// ==============================================================================
// FC_RouteFSM - Керування маршрутом (Mailbox Pattern v3.9)
// ==============================================================================
// Версія: 3.9.2
// Дата: 2026-02-27
// ==============================================================================
// ГАРАНТІЇ ЗУПИНКИ:
//   Нормальний STOP_OP:
//     STOPPING: CMD_STOP кожен цикл → STS_STOPPING→STS_IDLE →
//     allStopped → CMD_RELEASE_OWNER (ARB_OK) → ABORTED ✓
//
//   Аварія під час зупинки (STOPPING):
//     STS_FAULT → allStopped (FAULT рахується) →
//     CMD_RELEASE_OWNER (ARB_OK, FAULT дозволено) → ABORTED ✓
//
//   Enable_OK знімається під час зупинки (STOPPING):
//     STS_DISABLED + OwnerCur=NONE (механізм сам скинув) → allStopped →
//     CMD_RELEASE_OWNER → ARB_OWNER_BUSY (dummyOk) → ABORTED ✓
//
//   GlobalSafetyStop (механізм у STS_RUNNING):
//     CMD_STOP → Mechs[slot].Cmd=CMD_STOP → механізм → STS_STOPPING
//     CMD_RELEASE_OWNER → ARB_WRONG_STATUS (ще не IDLE) → ABORTED
//     Retry у ABORTED: STS_STOPPING→STS_IDLE → ARB_OK → OwnerCur=NONE ✓
//     (якщо апаратна безпека вбила живлення → STS_FAULT → ARB_OK ✓)
//
// АРХІТЕКТУРА:
//   FC_RouteFSM    — логіка переходів, послідовність кроків
//   FC_ArbiterMech — захоплення ownership, запис команди
//   FC_Noria/...   — виконання команди, зміна Status, аварії
//   FC_Route_Supervisor — Mailbox→RouteExecutor, виклик FSM, cleanup
// ==============================================================================

FUNCTION "FC_RouteFSM" : Void
{ S7_Optimized_Access := 'TRUE' }
VERSION : 3.7

VAR_INPUT
    RouteIdx          : USINT;            // ID маршруту (1..12)
    Cmd               : "UDT_RouteCmd";   // Команда та кроки маршруту
END_VAR

VAR_IN_OUT
    Mechs : ARRAY[0.."MECHS_COUNT"] OF "UDT_BaseMechanism";
    Fsm   : "UDT_RouteFsm";
END_VAR

VAR_OUTPUT
    Sts : "UDT_RouteStatus";
END_VAR

VAR_TEMP
    timeElapsed : BOOL;   // проміжний результат FC_TimeElapsedMs
    elapsedMs   : DINT;   // допоміжний вихід FC_TimeElapsedMs (ігнорується)
    nowTck      : DINT;   // допоміжний вихід FC_TimeElapsedMs (ігнорується)
    doAdvance   : BOOL;   // TRUE = виконати advance у STOPPING (після Phase A або Phase B)
END_VAR

BEGIN

    // =========================================================
    // Edge detection команд маршруту
    // =========================================================
    Fsm.startEdge  := (Cmd.RC_Cmd = "RT_CMD_START")   AND (Fsm.lastCmd <> "RT_CMD_START");
    Fsm.stopOpEdge := (Cmd.RC_Cmd = "RT_CMD_STOP_OP") AND (Fsm.lastCmd <> "RT_CMD_STOP_OP");
    Fsm.lastCmd    := Cmd.RC_Cmd;

    // =========================================================
    // Кількість кроків (з обмеженням)
    // =========================================================
    Fsm.stepCnt := USINT_TO_INT(Cmd.RC_StepCount);
    IF Fsm.stepCnt < 1  THEN Fsm.stepCnt := 1;  END_IF;
    IF Fsm.stepCnt > "ROUTE_MAX_STEPS" THEN Fsm.stepCnt := "ROUTE_MAX_STEPS"; END_IF;

    // Захист від неініціалізованого стану
    IF Fsm.RF_State = 0 THEN
        Fsm.RF_State := "ROUTE_STS_IDLE";
    END_IF;

    // =========================================================
    // Сканування механізмів: аварії та LocalManual
    // =========================================================
    Fsm.anyFault  := FALSE;
    Fsm.anyLocal  := FALSE;
    Fsm.safetyHit := FALSE;

    IF Fsm.stepCnt > 0 THEN
        FOR Fsm.i := 1 TO Fsm.stepCnt DO
            Fsm.slot := Cmd.RC_Steps[Fsm.i].RS_Slot;
            IF Fsm.slot > "MECHS_COUNT" THEN CONTINUE; END_IF;

            IF Mechs[Fsm.slot].FLTCode <> 0 THEN
                Fsm.anyFault := TRUE;
            END_IF;

            IF GlobalLocalManual OR Mechs[Fsm.slot].LocalManual THEN
                Fsm.anyLocal := TRUE;
            END_IF;

            IF Fsm.anyFault AND Fsm.anyLocal THEN EXIT; END_IF;
        END_FOR;
    END_IF;

    // =========================================================
    // АВАРІЙНА ЗУПИНКА (GlobalSafetyStop) — найвищий пріоритет
    // =========================================================
    // Послідовність для кожного механізму:
    //   1. CMD_STOP       — наказ зупинитись негайно (незалежно від послідовності)
    //                       ARB_OK → Mechs[slot].Cmd = CMD_STOP ✓
    //                       ARB_OWNER_BUSY → не наш механізм, не критично
    //                       ARB_LOCAL_MANUAL → оператор сам відповідає
    //   2. CMD_RELEASE_OWNER — спроба звільнити власника (best effort)
    //                       ARB_WRONG_STATUS якщо ще RUNNING/STOPPING → retry у ABORTED
    //
    // Чому не чекаємо STS_IDLE перед CMD_RELEASE_OWNER:
    //   Safety stop = негайно, без очікування. Механізм зупиниться сам
    //   (STS_STOPPING→STS_IDLE або апаратна безпека→STS_FAULT).
    //   Retry у ABORTED звільнить ownership коли механізм зупиниться.
    // =========================================================
    IF GlobalSafetyStop THEN
        Fsm.safetyHit := TRUE;

        IF Fsm.stepCnt > 0 THEN
            FOR Fsm.i := 1 TO Fsm.stepCnt DO
                Fsm.slot := Cmd.RC_Steps[Fsm.i].RS_Slot;
                IF Fsm.slot > "MECHS_COUNT" THEN CONTINUE; END_IF;

                // КРОК 1: Зупинити механізм
                Fsm.dummyOk := "FC_ArbiterMech"(
                    OwnerReq   := "OWNER_ROUTE",
                    OwnerReqId := USINT_TO_UINT(RouteIdx),
                    ReqCmd     := "CMD_STOP",
                    ReqParam1  := 0,
                    M          := Mechs[Fsm.slot]
                );

                // КРОК 2: Звільнити власника (best effort)
                // Якщо STS_RUNNING/STOPPING → ARB_WRONG_STATUS → retry у ABORTED
                Fsm.dummyOk := "FC_ArbiterMech"(
                    OwnerReq   := "OWNER_ROUTE",
                    OwnerReqId := USINT_TO_UINT(RouteIdx),
                    ReqCmd     := "CMD_RELEASE_OWNER",
                    ReqParam1  := 0,
                    M          := Mechs[Fsm.slot]
                );

            END_FOR;
        END_IF;

        Fsm.RF_State      := "ROUTE_STS_ABORTED";
        Fsm.RF_ResultCode := "ROUTE_ABRT_BY_SAFETY";
    END_IF;

    // =========================================================
    // FSM маршруту
    // =========================================================
    IF NOT Fsm.safetyHit THEN

        // --------------------------------------------------------
        // IDLE
        // --------------------------------------------------------
        IF Fsm.RF_State = "ROUTE_STS_IDLE" THEN

            IF Fsm.startEdge THEN
                Fsm.RF_ResultCode   := 0;
                Fsm.RF_AbortLatched := 0;
                Fsm.RF_ActiveStep   := 1;  // 1-based: перший крок [1]
                Fsm.RF_StepSts      := "STEP_STS_IDLE";
                Fsm.RF_State        := "ROUTE_STS_VALIDATING";
            END_IF;

        // --------------------------------------------------------
        // VALIDATING
        // --------------------------------------------------------
        ELSIF Fsm.RF_State = "ROUTE_STS_VALIDATING" THEN

            IF Fsm.stepCnt <= 0 THEN
                Fsm.RF_State      := "ROUTE_STS_REJECTED";
                Fsm.RF_ResultCode := "ROUTE_REJ_BY_CONTRACT";

            ELSE
                FOR Fsm.i := 1 TO Fsm.stepCnt DO
                    Fsm.slot   := Cmd.RC_Steps[Fsm.i].RS_Slot;
                    Fsm.stepOk := TRUE;

                    // Контракт: RS_Slot (перша перевірка — до будь-якого Mechs[slot])
                    IF Fsm.slot > "MECHS_COUNT" THEN
                        Fsm.stepOk := FALSE;
                    END_IF;

                    // Контракт: RS_Action
                    IF (Cmd.RC_Steps[Fsm.i].RS_Action <> "RS_ACT_START")
                       AND (Cmd.RC_Steps[Fsm.i].RS_Action <> "RS_ACT_STOP") THEN
                        Fsm.stepOk := FALSE;
                    END_IF;

                    // Контракт: RS_Wait
                    IF (Cmd.RC_Steps[Fsm.i].RS_Wait <> "RS_WAIT_RUNNING")
                       AND (Cmd.RC_Steps[Fsm.i].RS_Wait <> "RS_WAIT_STOPPED") THEN
                        Fsm.stepOk := FALSE;
                    END_IF;

                    // Контракт: RS_Action + RS_Wait сумісність
                    // RS_ACT_STOP + RS_WAIT_RUNNING: після CMD_STOP механізм іде
                    // STOPPING→IDLE і ніколи не повернеться у STS_RUNNING →
                    // крок ніколи не завершиться → маршрут зависає в RUNNING.
                    IF (Cmd.RC_Steps[Fsm.i].RS_Action = "RS_ACT_STOP")
                       AND (Cmd.RC_Steps[Fsm.i].RS_Wait = "RS_WAIT_RUNNING") THEN
                        Fsm.stepOk := FALSE;
                    END_IF;

                    IF NOT Fsm.stepOk THEN
                        Fsm.RF_State      := "ROUTE_STS_REJECTED";
                        Fsm.RF_ResultCode := "ROUTE_REJ_BY_CONTRACT";
                        EXIT;

                    ELSIF Mechs[Fsm.slot].OwnerCur <> "OWNER_NONE" THEN
                        Fsm.RF_State      := "ROUTE_STS_REJECTED";
                        Fsm.RF_ResultCode := "ROUTE_REJ_BY_OWNER";
                        EXIT;

                    ELSIF (NOT Mechs[Fsm.slot].Enable_OK)
                          OR GlobalLocalManual
                          OR Mechs[Fsm.slot].LocalManual
                          OR (Mechs[Fsm.slot].FLTCode <> 0) THEN
                        Fsm.RF_State      := "ROUTE_STS_REJECTED";
                        Fsm.RF_ResultCode := "ROUTE_REJ_NOT_READY";
                        EXIT;
                    END_IF;

                END_FOR;

                IF Fsm.RF_State = "ROUTE_STS_VALIDATING" THEN
                    Fsm.RF_State := "ROUTE_STS_STARTING";
                END_IF;
            END_IF;

        // --------------------------------------------------------
        // STARTING — атомарне захоплення всіх механізмів
        // --------------------------------------------------------
        ELSIF Fsm.RF_State = "ROUTE_STS_STARTING" THEN

            Fsm.lockOkAll := TRUE;

            IF Fsm.stepCnt > 0 THEN
                FOR Fsm.i := 1 TO Fsm.stepCnt DO
                    Fsm.slot := Cmd.RC_Steps[Fsm.i].RS_Slot;

                    // CMD_SET_OWNER_SCADA = захопити власника без виконання команди
                    Fsm.lockOkOne := "FC_ArbiterMech"(
                        OwnerReq   := "OWNER_ROUTE",
                        OwnerReqId := USINT_TO_UINT(RouteIdx),
                        ReqCmd     := "CMD_SET_OWNER_SCADA",
                        ReqParam1  := 0,
                        M          := Mechs[Fsm.slot]
                    );

                    IF Fsm.lockOkOne <> "ARB_OK" THEN
                        Fsm.lockOkAll := FALSE;
                    END_IF;
                END_FOR;
            ELSE
                Fsm.lockOkAll := FALSE;
            END_IF;

            IF NOT Fsm.lockOkAll THEN
                // Відкат: звільнити вже захоплені механізми.
                // Механізми ще у IDLE (не запускались) → CMD_RELEASE_OWNER пройде.
                // Механізм що не захопився → ARB_OWNER_BUSY → dummyOk.
                IF Fsm.stepCnt > 0 THEN
                    FOR Fsm.i := 1 TO Fsm.stepCnt DO
                        Fsm.slot := Cmd.RC_Steps[Fsm.i].RS_Slot;

                        Fsm.dummyOk := "FC_ArbiterMech"(
                            OwnerReq   := "OWNER_ROUTE",
                            OwnerReqId := USINT_TO_UINT(RouteIdx),
                            ReqCmd     := "CMD_RELEASE_OWNER",
                            ReqParam1  := 0,
                            M          := Mechs[Fsm.slot]
                        );
                    END_FOR;
                END_IF;

                Fsm.RF_State      := "ROUTE_STS_REJECTED";
                Fsm.RF_ResultCode := "ROUTE_REJ_BY_OWNER";

            ELSE
                Fsm.RF_State := "ROUTE_STS_RUNNING";
            END_IF;

        // --------------------------------------------------------
        // RUNNING — виконання кроків по черзі
        // --------------------------------------------------------
        ELSIF Fsm.RF_State = "ROUTE_STS_RUNNING" THEN

            // --- Умови переривання (перевіряються до виконання кроку) ---
            IF Fsm.stopOpEdge THEN
                Fsm.RF_AbortLatched := "ROUTE_ABRT_BY_OPERATOR";
                Fsm.RF_ActiveStep   := INT_TO_USINT(Fsm.stepCnt);  // 1-based: останній крок [stepCnt]
                Fsm.stepPause       := FALSE;
                Fsm.RF_State        := "ROUTE_STS_STOPPING";

            ELSIF Fsm.anyLocal THEN
                Fsm.RF_AbortLatched := "ROUTE_ABRT_BY_LOCAL";
                Fsm.RF_ActiveStep   := INT_TO_USINT(Fsm.stepCnt);  // 1-based
                Fsm.stepPause       := FALSE;
                Fsm.RF_State        := "ROUTE_STS_STOPPING";

            ELSIF Fsm.anyFault THEN
                Fsm.RF_AbortLatched := "ROUTE_ABRT_BY_FAULT";
                Fsm.RF_ActiveStep   := INT_TO_USINT(Fsm.stepCnt);  // 1-based
                Fsm.stepPause       := FALSE;
                Fsm.RF_State        := "ROUTE_STS_STOPPING";

            ELSE
                // --- Фаза B паузи або виконання поточного кроку ---
                IF Fsm.stepPause THEN
                    // ── Фаза B: пауза між кроками ────────────────────────────
                    // Крок виконано, механізм досягнув цільового стану.
                    // Нових команд не надсилаємо — чекаємо RS_TimeoutMs.
                    Fsm.stepIdx := USINT_TO_INT(Fsm.RF_ActiveStep);
                    timeElapsed := "FC_TimeElapsedMs"(
                            StartTck  := Fsm.stepPauseTck,
                            TimeoutMs := Cmd.RC_Steps[Fsm.stepIdx].RS_TimeoutMs,
                            ElapsedMs => elapsedMs,
                            NowTck    => nowTck);
                    IF timeElapsed THEN
                        Fsm.stepPause     := FALSE;
                        Fsm.RF_ActiveStep := Fsm.RF_ActiveStep + 1;
                        Fsm.RF_StepSts    := "STEP_STS_DONE";
                    END_IF;

                ELSE
                    // ── Фаза A: виконання поточного кроку ────────────────────
                    Fsm.stepIdx := USINT_TO_INT(Fsm.RF_ActiveStep);

                    IF Fsm.stepIdx > Fsm.stepCnt THEN
                        // Всі кроки виконано — залишаємось у RUNNING.
                        // Механізми залишаються під Owner=ROUTE.
                        // SCADA бачить ResultCode=200 → маршрут активний.
                        Fsm.RF_ResultCode := "ROUTE_OK_RUNNING";  // 200

                    ELSE
                        Fsm.slot := Cmd.RC_Steps[Fsm.stepIdx].RS_Slot;

                        // Видати команду поточного кроку через арбітр
                        IF Cmd.RC_Steps[Fsm.stepIdx].RS_Action = "RS_ACT_START" THEN
                            Fsm.cmdOk := "FC_ArbiterMech"(
                                OwnerReq   := "OWNER_ROUTE",
                                OwnerReqId := USINT_TO_UINT(RouteIdx),
                                ReqCmd     := "CMD_START",
                                ReqParam1  := Cmd.RC_Steps[Fsm.stepIdx].RS_StartParam,
                                M          := Mechs[Fsm.slot]
                            );
                        ELSE
                            Fsm.cmdOk := "FC_ArbiterMech"(
                                OwnerReq   := "OWNER_ROUTE",
                                OwnerReqId := USINT_TO_UINT(RouteIdx),
                                ReqCmd     := "CMD_STOP",
                                ReqParam1  := 0,
                                M          := Mechs[Fsm.slot]
                            );
                        END_IF;

                        IF Fsm.cmdOk <> "ARB_OK" THEN
                            // Арбітр відхилив команду → аварійна зупинка маршруту
                            Fsm.RF_AbortLatched := "ROUTE_ABRT_BY_OWNER";
                            Fsm.RF_ActiveStep   := INT_TO_USINT(Fsm.stepCnt);  // 1-based
                            Fsm.stepPause       := FALSE;
                            Fsm.RF_State        := "ROUTE_STS_STOPPING";

                        ELSE
                            Fsm.RF_StepSts := "STEP_STS_WORK";

                            // Перевірити умову завершення кроку.
                            // RS_TimeoutMs > 0 → Фаза B (пауза), інакше advance одразу.
                            IF Cmd.RC_Steps[Fsm.stepIdx].RS_Wait = "RS_WAIT_RUNNING" THEN
                                IF Mechs[Fsm.slot].Status = "STS_RUNNING" THEN
                                    IF Cmd.RC_Steps[Fsm.stepIdx].RS_TimeoutMs > 0 THEN
                                        timeElapsed := "FC_TimeElapsedMs"(
                                                           StartTck  := 0,
                                                           TimeoutMs := 0,
                                                           ElapsedMs => elapsedMs,
                                                           NowTck    => Fsm.stepPauseTck);
                                        Fsm.stepPause := TRUE;
                                    ELSE
                                        Fsm.RF_ActiveStep := Fsm.RF_ActiveStep + 1;
                                        Fsm.RF_StepSts    := "STEP_STS_DONE";
                                    END_IF;
                                END_IF;
                            ELSE  // RS_WAIT_STOPPED
                                IF Mechs[Fsm.slot].Status = "STS_IDLE" THEN
                                    IF Cmd.RC_Steps[Fsm.stepIdx].RS_TimeoutMs > 0 THEN
                                        timeElapsed := "FC_TimeElapsedMs"(
                                                           StartTck  := 0,
                                                           TimeoutMs := 0,
                                                           ElapsedMs => elapsedMs,
                                                           NowTck    => Fsm.stepPauseTck);
                                        Fsm.stepPause := TRUE;
                                    ELSE
                                        Fsm.RF_ActiveStep := Fsm.RF_ActiveStep + 1;
                                        Fsm.RF_StepSts    := "STEP_STS_DONE";
                                    END_IF;
                                END_IF;
                            END_IF;
                        END_IF;
                    END_IF;
                END_IF;
            END_IF;

        // --------------------------------------------------------
        // STOPPING — покрокова зупинка у зворотньому порядку з паузою
        // --------------------------------------------------------
        // RF_ActiveStep = поточний крок зупинки (stepCnt → 1).
        // Ініціалізується при вході з RUNNING (= stepCnt).
        //
        // Дві фази для кожного кроку:
        //   Фаза A (stepPause=FALSE): CMD_STOP кожен цикл → чекаємо зупинки.
        //     Зупинився + RS_TimeoutMs > 0 → stepPause:=TRUE (перейти у Фазу B).
        //     Зупинився + RS_TimeoutMs = 0 → doAdvance:=TRUE (advance одразу).
        //   Фаза B (stepPause=TRUE): чекаємо RS_TimeoutMs мс, CMD_STOP не надсилаємо.
        //     Час вийшов → stepPause:=FALSE, doAdvance:=TRUE.
        //
        //   Advance (doAdvance=TRUE):
        //     stepIdx > 1 → RF_ActiveStep-- (наступний крок у Фазі A)
        //     stepIdx = 1 → CMD_RELEASE_OWNER для всіх → ABORTED
        //
        // "Зупинений": STS_IDLE / STS_FAULT / STS_DISABLED / STS_LOCAL
        // "НЕ зупинений": STS_STARTING / STS_RUNNING / STS_STOPPING
        // --------------------------------------------------------
        ELSIF Fsm.RF_State = "ROUTE_STS_STOPPING" THEN

            IF Fsm.stepCnt > 0 THEN
                Fsm.stepIdx := USINT_TO_INT(Fsm.RF_ActiveStep);
                Fsm.slot    := Cmd.RC_Steps[Fsm.stepIdx].RS_Slot;
                doAdvance   := FALSE;

                IF Fsm.stepPause THEN
                    // ── Фаза B: пауза між кроками ────────────────────────────
                    // CMD_STOP не надсилаємо — механізм вже зупинений.
                    // Чекаємо RS_TimeoutMs мс. Час вийшов → doAdvance.
                    timeElapsed := "FC_TimeElapsedMs"(
                            StartTck  := Fsm.stepPauseTck,
                            TimeoutMs := Cmd.RC_Steps[Fsm.stepIdx].RS_TimeoutMs,
                            ElapsedMs => elapsedMs,
                            NowTck    => nowTck);
                    IF timeElapsed THEN
                        Fsm.stepPause := FALSE;
                        doAdvance     := TRUE;
                    END_IF;

                ELSE
                    // ── Фаза A: зупинка поточного механізму ─────────────────
                    // CMD_STOP (або StopParam) кожен цикл (рівневе керування)
                    IF Cmd.RC_Steps[Fsm.stepIdx].RS_StopParam <> 0 THEN
                        // Параметрична зупинка (напр., засувка у позицію CLOSED)
                        Fsm.dummyOk := "FC_ArbiterMech"(
                            OwnerReq   := "OWNER_ROUTE",
                            OwnerReqId := USINT_TO_UINT(RouteIdx),
                            ReqCmd     := "CMD_START",
                            ReqParam1  := Cmd.RC_Steps[Fsm.stepIdx].RS_StopParam,
                            M          := Mechs[Fsm.slot]
                        );
                    ELSE
                        Fsm.dummyOk := "FC_ArbiterMech"(
                            OwnerReq   := "OWNER_ROUTE",
                            OwnerReqId := USINT_TO_UINT(RouteIdx),
                            ReqCmd     := "CMD_STOP",
                            ReqParam1  := 0,
                            M          := Mechs[Fsm.slot]
                        );
                    END_IF;

                    // Перевірка: чи поточний механізм зупинився
                    IF (Mechs[Fsm.slot].Status <> "STS_STARTING")
                    AND (Mechs[Fsm.slot].Status <> "STS_RUNNING")
                    AND (Mechs[Fsm.slot].Status <> "STS_STOPPING") THEN

                        IF Cmd.RC_Steps[Fsm.stepIdx].RS_TimeoutMs > 0 THEN
                            // Запустити паузу (Фаза B): захопити поточний час
                            timeElapsed := "FC_TimeElapsedMs"(
                                               StartTck  := 0,
                                               TimeoutMs := 0,
                                               ElapsedMs => elapsedMs,
                                               NowTck    => Fsm.stepPauseTck);
                            Fsm.stepPause := TRUE;
                        ELSE
                            doAdvance := TRUE;  // RS_TimeoutMs = 0: advance одразу
                        END_IF;

                    END_IF;
                END_IF;

                // ── Advance ───────────────────────────────────────────────────
                // Виконується ТІЛЬКИ коли явно встановлено doAdvance:
                //   - Phase A: механізм зупинився + RS_TimeoutMs = 0
                //   - Phase B: таймер спрацював
                IF doAdvance THEN
                    IF Fsm.stepIdx > 1 THEN
                        // Перейти до попереднього кроку (Фаза A)
                        Fsm.RF_ActiveStep := Fsm.RF_ActiveStep - 1;

                    ELSE
                        // Всі механізми зупинено → CMD_RELEASE_OWNER + ABORTED
                        // ARB_WRONG_STATUS (STS_DISABLED/LOCAL) → retry у ABORTED
                        FOR Fsm.i := 1 TO Fsm.stepCnt DO
                            Fsm.slot := Cmd.RC_Steps[Fsm.i].RS_Slot;
                            Fsm.dummyOk := "FC_ArbiterMech"(
                                OwnerReq   := "OWNER_ROUTE",
                                OwnerReqId := USINT_TO_UINT(RouteIdx),
                                ReqCmd     := "CMD_RELEASE_OWNER",
                                ReqParam1  := 0,
                                M          := Mechs[Fsm.slot]
                            );
                        END_FOR;

                        IF Fsm.RF_AbortLatched = 0 THEN
                            Fsm.RF_AbortLatched := "ROUTE_ABRT_BY_OPERATOR";
                        END_IF;
                        Fsm.RF_ResultCode := Fsm.RF_AbortLatched;
                        Fsm.RF_State      := "ROUTE_STS_ABORTED";
                    END_IF;
                END_IF;

            ELSE
                // stepCnt = 0 (не повинно траплятись після STARTING) → відразу ABORTED
                IF Fsm.RF_AbortLatched = 0 THEN
                    Fsm.RF_AbortLatched := "ROUTE_ABRT_BY_OPERATOR";
                END_IF;
                Fsm.RF_ResultCode := Fsm.RF_AbortLatched;
                Fsm.RF_State      := "ROUTE_STS_ABORTED";
            END_IF;

        // --------------------------------------------------------
        // REJECTED / ABORTED
        // --------------------------------------------------------
        ELSIF (Fsm.RF_State = "ROUTE_STS_REJECTED")
           OR (Fsm.RF_State = "ROUTE_STS_ABORTED") THEN

            // ---------------------------------------------------------
            // RETRY CMD_RELEASE_OWNER — вирішення застряглого ownership.
            //
            // Типовий сценарій після GlobalSafetyStop:
            //   Цикл N:     CMD_STOP → OK, CMD_RELEASE_OWNER → ARB_WRONG_STATUS
            //   Цикли N+1..: retry кожен цикл поки механізм зупиняється
            //   STS_STOPPING → STS_IDLE → ARB_OK → OwnerCur=NONE ✓
            //   (або апаратна безпека → STS_FAULT → ARB_OK ✓)
            //
            // Умова IF: тільки наші механізми (OwnerCur/OwnerCurId перевіряємо).
            // Якщо вже NONE — умова FALSE, виклик не відбувається.
            // ---------------------------------------------------------
            IF Fsm.stepCnt > 0 THEN
                FOR Fsm.i := 1 TO Fsm.stepCnt DO
                    Fsm.slot := Cmd.RC_Steps[Fsm.i].RS_Slot;

                    IF (Mechs[Fsm.slot].OwnerCur   =  "OWNER_ROUTE")
                   AND (Mechs[Fsm.slot].OwnerCurId =  USINT_TO_UINT(RouteIdx)) THEN

                        Fsm.dummyOk := "FC_ArbiterMech"(
                            OwnerReq   := "OWNER_ROUTE",
                            OwnerReqId := USINT_TO_UINT(RouteIdx),
                            ReqCmd     := "CMD_RELEASE_OWNER",
                            ReqParam1  := 0,
                            M          := Mechs[Fsm.slot]
                        );
                        // ARB_OK           → OwnerCur = NONE ✓
                        // ARB_WRONG_STATUS → ще не IDLE/FAULT, retry наступний цикл
                    END_IF;

                END_FOR;
            END_IF;

            // Re-start: startEdge → прямо у VALIDATING (без проміжного IDLE).
            // Supervisor вже скопіював кроки у RouteExecutor (Cleanup захищений processedRouteId).
            // Якщо механізми ще OWNER_ROUTE (ABORTED-retry не завершено) →
            //   VALIDATING поверне ROUTE_REJ_BY_OWNER (коректна поведінка).
            IF Fsm.startEdge THEN
                Fsm.RF_ResultCode   := 0;
                Fsm.RF_AbortLatched := 0;
                Fsm.RF_ActiveStep   := 1;  // 1-based: перший крок [1]
                Fsm.RF_StepSts      := "STEP_STS_IDLE";
                Fsm.RF_State        := "ROUTE_STS_VALIDATING";

            // Перехід у IDLE коли Supervisor очистить команду (RT_CMD_NONE)
            ELSIF Cmd.RC_Cmd = "RT_CMD_NONE" THEN
                Fsm.RF_State := "ROUTE_STS_IDLE";
            END_IF;

        ELSE
            // Невідомий стан — скидаємо
            Fsm.RF_State := "ROUTE_STS_IDLE";
        END_IF;

    END_IF;

    // =========================================================
    // Вихідний статус
    // =========================================================
    Sts.RS_State      := Fsm.RF_State;
    Sts.RS_ResultCode := Fsm.RF_ResultCode;
    Sts.RS_ActiveStep := Fsm.RF_ActiveStep;
    Sts.RS_StepSts    := Fsm.RF_StepSts;

END_FUNCTION
